FUNCTION_BLOCK FB_GantryXY EXTENDS FB_PackML_BaseModule
VAR
    // Sub module definitions here

    // List of sub modules
    ipSubModules_Init : ARRAY[1..Parameters_PackML_Base.MAX_NO_OF_SUBMODULES] OF I_PackML_BaseModule := [];

    // Component definitions here
    AxisX       		: FB_Component_BasicAxis 		:= (Name := 'AxisX');
    AxisY    			: FB_Component_BasicAxis 		:= (Name := 'AxisY');
    GantryCylinder		: FB_GantryXYCylinder			:= (Name := 'Cylinder');

    //Alarms for this module
    GantryAlarms : ARRAY[1..GANTRY_ALARM_COUNT] OF FB_TcAlarm;

	//IO
	PositionSensorX :BOOL;
	PositionSensorY :BOOL;

	AxisXHomingComplete :BOOL;
	AxisYHomingComplete :BOOL;

END_VAR

VAR CONSTANT
    //Alarms
    GANTRY_ALARM_COUNT : INT := 5;
END_VAR

//! @summary This method contains code which will execute when this PackML module is in the <b>Aborted</b> state
METHOD PROTECTED Aborted

(*! <description> <b>The base implementation of this method is empty. User must override this method to provide functionality.</b>
<table> 
	<tr>
		<th> Previous State </th>
		<th> Transition In </th>
		<th> Transition Out </th>
		<th> Next State  </th> 
	</tr>
	<tr>
		<td> Aborting </td>
		<td> State Complete <i>(Aborting)</i></td> 
		<td> Clear Command </td>
		<td> Clearing </td> 
	</tr>
</table>
This method is called as required by <c>StateControl()</c>
</description> 

*)
END_METHOD

//! @summary This method contains code which will execute when this PackML module is in the <b>Clearing</b> state
METHOD PROTECTED Clearing
VAR
	i				: UDINT;
	SubModulesReady : BOOL := TRUE;
END_VAR

(*! <description> <b>Note:</b> The <i>Clear</i> command can also be thought of as a <i>fault reset</i> depite the ambiguity in the naming of the <i>Reset</i> state. 
<table> 
	<tr>
		<th> Previous State </th>
		<th> Transition In </th>
		<th> Transition Out </th>
		<th> Next State  </th> 
	</tr>
	<tr>
		<td> Aborted </td>
		<td> Clear Command </td> 
		<td> State Complete </td>
		<td> Stopped </td> 
	</tr>
</table>
This method is called as required by <c>StateControl()</c>
</description> 

*)
CASE SequenceState OF
    0:
        NoStateTasksToComplete := FALSE;
        SequenceState          := SequenceState + 10;
    10:
        //Reset any alarms that get latched
        GantryAlarms[E_Gantry.StartTimeout].Clear(0,0);
        SequenceState := SequenceState + 10;
    20:
        // Enable here
        AxisX.Enable();
		AxisY.Enable();

        // Check enabled here
        IF AxisX.Enabled AND AxisY.Enabled THEN
            SequenceState := SequenceState + 10;
        END_IF
    30:
        StateTasksComplete := TRUE;
END_CASE

SUPER^.Clearing();
END_METHOD

METHOD PROTECTED CreateEvents
VAR_INPUT
END_VAR
// Add your event creation here
F_CreateAllEventsInClass(Alarms     := GantryAlarms,
                         ClassSize  := SIZEOF(TC_EVENTS.Gantry),
                         pInitEvent := ADR(TC_EVENTS.Gantry.InitReferenceEvent),
                         Prefix     := _Name);

// Super call to base
SUPER^.CreateEvents();
END_METHOD

METHOD CyclicLogic
VAR_INPUT
END_VAR
IF NOT _InitComplete THEN
    _InitComplete := Initialize();
    RETURN;
END_IF

SUPER^.CyclicLogic();

//Set the current alarm severity for this module
_CurrentAlarmSeverity := F_GetMaxSeverityRaised(Alarms := GantryAlarms, CurrentSeverity := _CurrentAlarmSeverity);

//Simulate Alarm Messaging
END_METHOD

//! @summary This method contains code which will execute when this PackML module is in the <b>Execute</b> state
METHOD PROTECTED Execute

(*! <description> <b>The base implementation of this method is empty. User must override this method to provide functionality.</b>
<table> 
	<tr>
		<th> Previous State </th>
		<th> Transition In </th>
		<th> Transition Out </th>
		<th> Next State  </th> 
	</tr>
	<tr>
		<td> Starting<b>-or-</b>Unholding <b>-or-</b>Unsuspending</td>
		<td> State Complete<i>(Starting<b>-or-</b>Unholding<b>-or-</b>Unsuspending)</i></td> 
		<td> State Complete<b>-or-</b>Hold Command<b>-or-</b>Suspend Command</td>
		<td> Completing<b>-or-</b>Holding<b>-or-</b>Suspending</td>
	</tr>
</table>
This method is called as required by <c>StateControl()</c>
</description> 

*)
END_METHOD

//! @summary This method contains code which will execute when this PackML module is in the <b>Idle</b> state
METHOD PROTECTED Idle

(*! <description> <b>The base implementation of this method is empty. User must override this method to provide functionality.</b>
<table> 
	<tr>
		<th> Previous State </th>
		<th> Transition In </th>
		<th> Transition Out </th>
		<th> Next State  </th> 
	</tr>
	<tr>
		<td> Resetting </td>
		<td> State Complete <i>(Resetting)</i></td> 
		<td> Start Command </td>
		<td> Starting </td> 
	</tr>
</table>
This method is called as required by <c>StateControl()</c>
</description> 

*)
END_METHOD

//! @summary Basic module initialization logic
METHOD PROTECTED Initialize : BOOL;
VAR
    i                        : UDINT;
    varInfo                  : __SYSTEM.VAR_INFO;
    AllSubUnitsInitialized   : BOOL := TRUE;
    AllComponentsInitialized : BOOL := TRUE;
END_VAR

//! @description This method is called by <c>CyclicLogic()</c> as required
Initialize := FALSE;
CASE DescendantSequenceState OF
    0:
		RegisterComponent(AxisX);
		RegisterComponent(AxisY);		
		RegisterComponent(GantryCylinder);
		
        _LogModeChanges         := FALSE;
        _LogStateChanges        := FALSE;
        DescendantSequenceState := DescendantSequenceState + 10;
    10:
        DescendantSequenceState := DescendantSequenceState + 10;
    20:
        //Copy Mode names
        FOR i := 1 TO 3 DO
            ModeNames[i] := F_UnitModeToString(UDINT_TO_DINT(i));
        END_FOR

        DescendantSequenceState := DescendantSequenceState + 10;
    30:
        //Call the Super
        IF SUPER^.Initialize() THEN
            DescendantSequenceState := DescendantSequenceState + 10;
        END_IF
    40:
        Initialize := TRUE;
END_CASE
END_METHOD

METHOD PROTECTED Starting
VAR
	i				: UDINT;
	SubModulesReady : BOOL := TRUE;
END_VAR
CASE _CurrentMode OF

	//=================================PRODUCTION MODE==================================
	E_PMLUnitMode.ePMLUnitMode_Production:
		CASE SequenceState OF
			0:
				
				NoStateTasksToComplete := FALSE;

					AxisX.Home();
					AxisY.Home();
					SequenceState := SequenceState + 10;

			10:
				StateTasksComplete := TRUE;


		END_CASE

	//=================================MAINTENANCE & MANUAL MODE==================================
	E_PMLUnitMode.ePMLUnitMode_Maintenance, E_PMLUnitMode.ePMLUnitMode_Manual:
		;
END_CASE

SUPER^.Starting();
END_METHOD

//! @summary This method contains code which will execute when this PackML module is in the <b>Stopped</b> state
METHOD PROTECTED Stopped

(*! <description> <b>The base implementation of this method is empty. User must override this method to provide functionality.</b>
<table> 
	<tr>
		<th> Previous State </th>
		<th> Transition In </th>
		<th> Transition Out </th>
		<th> Next State  </th> 
	</tr>
	<tr>
		<td> Stopping<b>-or-</b>Clearing </td>
		<td> State Complete <i>(Stopping<b>-or-</b>Clearing)</i></td> 
		<td> Reset Command </td>
		<td> Resetting </td> 
	</tr>
</table>
This method is called as required by <c>StateControl()</c>
</description> 

*)
END_METHOD

END_FUNCTION_BLOCK

(* stored: Version 1.1.0.1
   POU FB_GantryXY: Id {496b17f1-4b0a-4954-89f4-eec9ef72b2f5}, SpecialFunc None
   Folder GantryXYStates: Id {83d122fa-7c6a-0e7c-1bbf-3cae8b533243}
   Method Aborted: Id {7a5dcb3e-2759-094f-1862-434dd6d18864}
   Method Clearing: Id {fd669db8-130b-0177-023d-92edf1bab84d}
   Method CreateEvents: Id {4ec0ace2-c308-44b2-84a1-60ba649bd547}
   Method CyclicLogic: Id {02def406-fced-425b-89cd-43b7d8052b02}
   Method Execute: Id {8bbd73eb-f81f-0125-146b-eb6c70f49230}
   Method Idle: Id {0745b186-03c9-09b7-0039-cfbaac37c0d8}
   Method Initialize: Id {b4a0fd62-4385-4420-ae43-9bea35a3f798}
   Method Starting: Id {7539693f-63b4-09d4-0a7e-598ba148d1a2}
   Method Stopped: Id {4651aaa0-3084-0692-39f1-f4fedfe67bb4} *)
